FUNCTION_BLOCK PairTagTask EXTENDS TcoCore.TcoRemoteTask
VAR
	
	_key: STRING;
	_assignedValue : STRING;	
	_answerInstruction : STRING(254);
	_answer: TagsPairing;
	{attribute 'hide'}
	_answerClean: TagsPairing;
	_mode: eTagPairingMode;
END_VAR

SUPER^();

PROPERTY Answer : TagsPairing
GET
Answer:=_answer;
END_GET
END_PROPERTY

PROPERTY AnswerInstruction : string
GET
VAR
	retVal: STRING;
END_VAR
AnswerInstruction :=_answerInstruction;
END_GET
END_PROPERTY

(*~
	<docu>
		<summary>
			Restores this instance to the Ready state. Can be called explicitly or from within one of the restore mechanisms.
			<para>
				See also <see cref="PlcDocu.TcoCore.TcoTask.AutoRestorable()"/>
			</para>
		</summary>			
	</docu>	
~*)
METHOD Restore : ITcoRestorable
SUPER^.Restore();
_answer:=_answerClean;
END_METHOD

METHOD Run : REFERENCE TO PairTagTask
VAR_INPUT
	(*~
	<docu>
		<summary>
			The mode is type of operation to be done by invoking  this remote task.(GetTag,CreateTag...)
		</summary>						
	</docu>	
	~*)
	inMode :eTagPairingMode;
	(*~
	<docu>
		<summary>
			The Key is ID  of the tag's Uid on which assigned value will be found . 	
		</summary>						
	</docu>	
	~*)
	inKey : STRING;
		(*~
	<docu>
		<summary>
			The AAssignedValue is user defined additional value, this value provide  better undersanding identification of carriers . 	
		</summary>						
	</docu>	
	~*)
	inAssignedValue : STRING;
	
END_VAR
THIS^._key := inKey;
THIS^._mode := inMode;
THIS^._assignedValue := inAssignedValue;


Run REF= THIS^;
END_METHOD

END_FUNCTION_BLOCK

(* stored: Version 1.1.0.1
   POU PairTagTask: Id {b083ca0f-7862-4042-9ba0-9233a2104f8e}, SpecialFunc None
   Property Answer: Id {8dbbb230-6fd8-4cd9-a004-ea5f80e0b2d6}
   Get Get: Id {b2c02d2a-2ee9-4b05-bc9f-52cb6497fa69}
   Property AnswerInstruction: Id {38bbcf52-7bdf-400e-bbe2-be224e427c46}
   Get Get: Id {f8ea9d96-50e2-4901-9759-3031dac03323}
   Method Restore: Id {771560ea-d503-408a-ae88-5ce69517fc8b}
   Method Run: Id {b1078f12-a7f9-4b35-95ef-8e26e435bc71} *)
